INTERFACE I_MotionBrake


METHOD ActivateBrake
END_METHOD


METHOD BrakeIsActivated : BOOL
END_METHOD


METHOD DeactivateBrake
END_METHOD

END_INTERFACE

(* stored: Version 1.1.0.1
   Itf I_MotionBrake: Id {9c73ed1c-5ca5-43f4-920f-de00f3960209}
   Method ActivateBrake: Id {98d792eb-0263-480f-94cd-8d0195ec52e5}
   Method BrakeIsActivated: Id {bd57112d-1890-48a0-aee6-60d268124525}
   Method DeactivateBrake: Id {b8bc6fae-b65d-4582-b262-72b4efdb8aeb} *)
